(* CoDeSys 2.3.9.50 project: 3D.pr6 *)
(* Libraries: STANDARD.LB6 5.6.98 12:03:02 *)

(* POU MAIN, LD *)
PROGRAM MAIN
VAR
	Start AT %IX0.0: BOOL;
	t1: TON;
	t2: TON;
	t3: TON;
	mixA AT %QX0.0: BOOL;
	mixB AT %QX0.1: BOOL;
	mixC AT %QX0.2: BOOL;
	MasterEnable AT %IX0.0: BOOL;
END_VAR
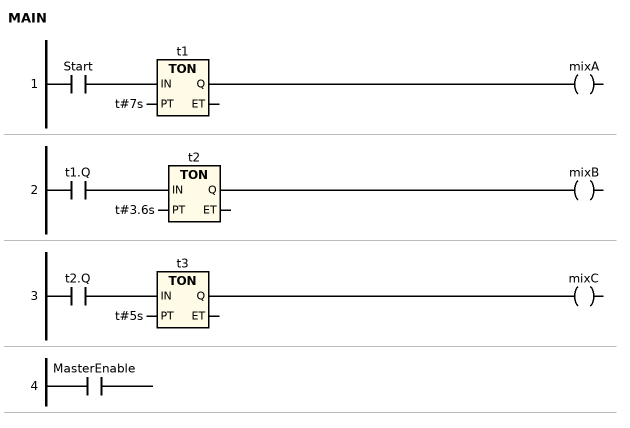
_LD_ (* Ladder Diagram *)
NETWORK 1
	[Start] - t1:TON(IN: *, PT: t#7s) --- (mixA)
NETWORK 2
	[t1.Q] - t2:TON(IN: *, PT: t#3.6s) --- (mixB)
NETWORK 3
	[t2.Q] - t3:TON(IN: *, PT: t#5s) --- (mixC)
NETWORK 4
	[MasterEnable]
_END_LD_
(* the same logic as Structured Text *)
(* Network 1 *)
t1(IN := Start, PT := t#7s);
mixA := t1.Q;
(* Network 2 *)
t2(IN := t1.Q, PT := t#3.6s);
mixB := t2.Q;
(* Network 3 *)
t3(IN := t2.Q, PT := t#5s);
mixC := t3.Q;
(* Network 4 *)
END_PROGRAM
